PROGRAM Prg_NonInstantFunc
VAR
	Buttons: ARRAY[1..4] OF BOOL;
	Temp: ARRAY[1..4] OF INT := [90, 20, 100, 75];
	OverLoad: ARRAY[1..4] OF BOOL;
	AnalogSensor: ARRAY[1..4] OF INT := [8, 0, 8, 0];
	Coils: ARRAY[1..4] OF BOOL;
	
	i: INT;
	
END_VAR

FOR i:=1 TO 4 BY 1 DO
	IF CheckFault(Overload:=OverLoad[i], MotorTemp:=Temp[i]) THEN
		Coils[i]:=FALSE;
	ELSIF Buttons[i] THEN
		Coils[i]:=TRUE;
	ELSE
		Coils[i]:=FALSE;		
	END_IF
END_FOR

END_PROGRAM

(* stored: Version 1.1.0.1, ProductVersion 3.1.4024.9
   POU Prg_NonInstantFunc: Id {314535fe-c8fe-41d5-b4c9-26aaffeb0411}, SpecialFunc None *)
